// Mitsubishi GX Works2 project: 往复式传送带   PLC: FX3U/FX3UC

PROGRAM MAIN
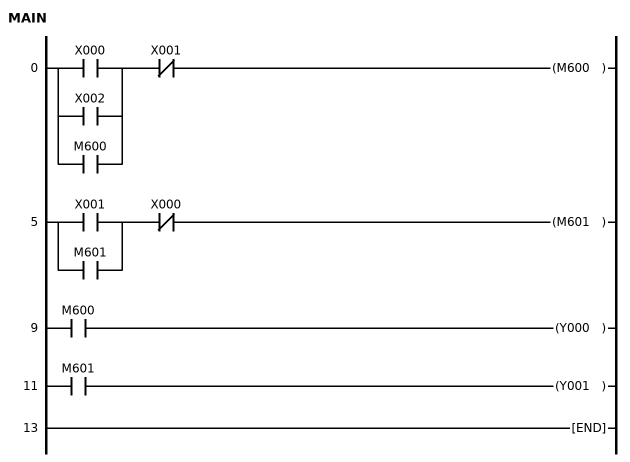
0     LD      X000
      OR      X002
      OR      M600
      ANI     X001
      OUT     M600
5     LD      X001
      OR      M601
      ANI     X000
      OUT     M601
9     LD      M600
      OUT     Y000
11    LD      M601
      OUT     Y001
13    END
END_PROGRAM
